Fanuc KAREL source: DISMOUNT_DEV.kl

PROGRAM T
%NOLOCKGROUP
VAR
 v0 : STRING[40]
 v1 : INTEGER
BEGIN
 DISMOUNT_DEV(v0, v1)
END T
